{attribute addProperty BoxType "AT2021-0250-0018"}
{attribute addProperty Id "CC_InputsAT %I*CC_Inputs_9818D8D8256320CC_OutputsAT %Q*CC_Outputs_AA78E99F256320WcStateAT %I*WcState_98A4DF7520.250InfoDataAT %I*InfoData_0BDED7BF144180"}
{attribute addProperty CRC "3298337665"}
{attribute addProperty SizeInBites "658"}
{attribute addProperty SizeInBytes "82.25"}
TYPE AT2021_BA5A9548 :
STRUCT
	{attribute addProperty Name "CC_Inputs"}
	CC_Inputs : CC_Inputs_9818D8D8;
	{attribute addProperty Name "CC_Outputs"}
	CC_Outputs : CC_Outputs_AA78E99F;
	{attribute addProperty Name "WcState"}
	WcState : WcState_98A4DF75;
	{attribute addProperty Name "InfoData"}
	InfoData : InfoData_0BDED7BF;
END_STRUCT
END_TYPE

(* stored: Version 1.2.0.0, ProductVersion 3.1.4024.9
   DUT AT2021_BA5A9548: Id {9de8251f-e8bf-4508-816f-53b4d648ac2a} *)
